(* Manages alarms *)

PROGRAM Alarm_Manager
  VAR_EXTERNAL
    Safety_OK : BOOL;
    Conveyor_Fault : BOOL;
    Mixer_Fault : BOOL;
    Packaging_Fault : BOOL;
    Pump_A_Fault : BOOL;
    Pump_B_Fault : BOOL;
    Discharge_Pump_Fault : BOOL;
    Inlet_Valve_Fault : BOOL;
    Ingredient_A_Valve_Fault : BOOL;
    Ingredient_B_Valve_Fault : BOOL;
    Discharge_Valve_Fault : BOOL;
    Batch : ST_BATCH;
    Temperature : REAL;
    Conveyor_Jam : BOOL;
    Batch_State_Code : INT;
    System_Reset : BOOL;
    Alarm_Acknowledge : BOOL;
  END_VAR
  VAR
    Safety_Alarm : ST_ALARM;
    Conveyor_Alarm : ST_ALARM;
    Mixer_Alarm : ST_ALARM;
    Packaging_Alarm : ST_ALARM;
    Pump_A_Alarm : ST_ALARM;
    Pump_B_Alarm : ST_ALARM;
    Discharge_Pump_Alarm : ST_ALARM;
    Inlet_Valve_Alarm : ST_ALARM;
    Ingredient_A_Valve_Alarm : ST_ALARM;
    Ingredient_B_Valve_Alarm : ST_ALARM;
    Discharge_Valve_Alarm : ST_ALARM;
    Conveyor_Jam_Alarm : ST_ALARM;
    Batch_Fault_Alarm : ST_ALARM;
    Temperature_Alarm : ST_ALARM;
    Any_Alarm : BOOL;
  END_VAR

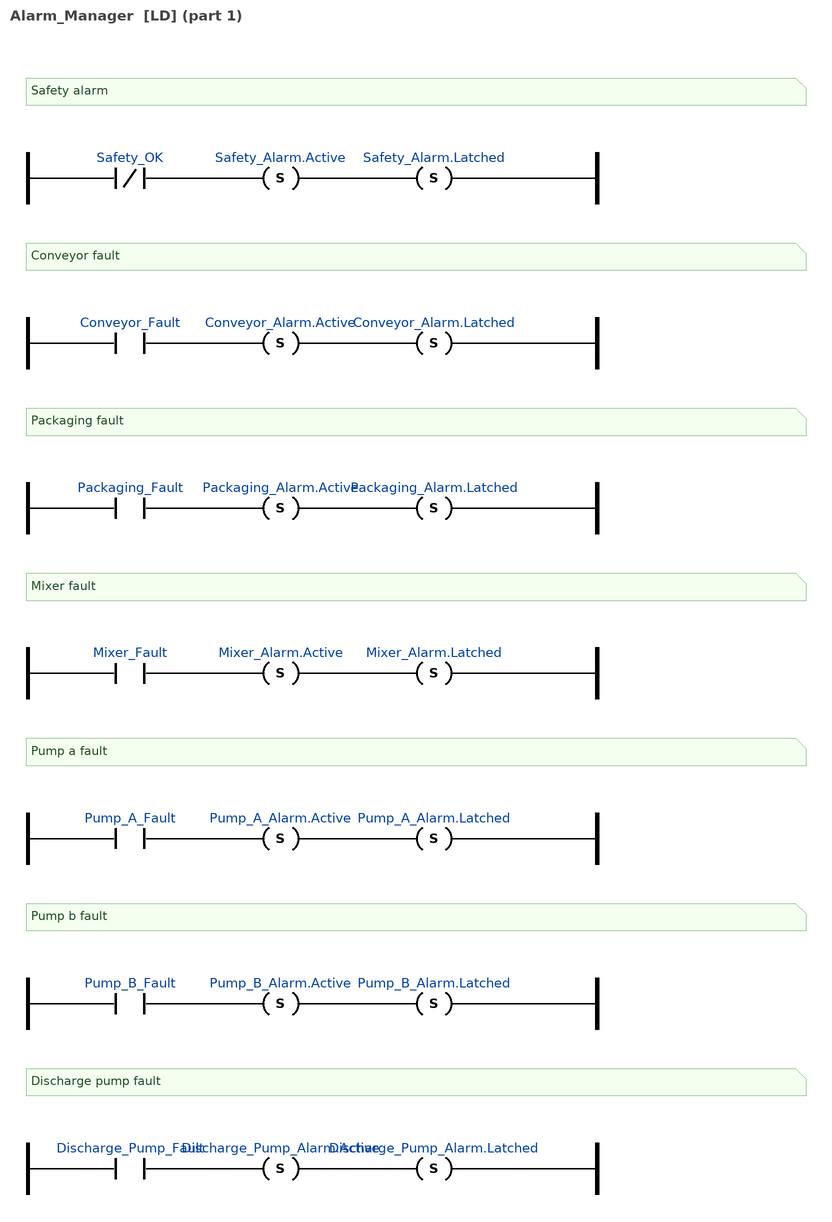
(* LD diagram, written out as Structured Text *)
(* Safety alarm *)
IF NOT Safety_OK THEN Safety_Alarm.Active := TRUE; END_IF;
IF NOT Safety_OK THEN Safety_Alarm.Latched := TRUE; END_IF;
(* Conveyor fault *)
IF Conveyor_Fault THEN Conveyor_Alarm.Active := TRUE; END_IF;
IF Conveyor_Fault THEN Conveyor_Alarm.Latched := TRUE; END_IF;
(* Packaging fault *)
IF Packaging_Fault THEN Packaging_Alarm.Active := TRUE; END_IF;
IF Packaging_Fault THEN Packaging_Alarm.Latched := TRUE; END_IF;
(* Mixer fault *)
IF Mixer_Fault THEN Mixer_Alarm.Active := TRUE; END_IF;
IF Mixer_Fault THEN Mixer_Alarm.Latched := TRUE; END_IF;
(* Pump a fault *)
IF Pump_A_Fault THEN Pump_A_Alarm.Active := TRUE; END_IF;
IF Pump_A_Fault THEN Pump_A_Alarm.Latched := TRUE; END_IF;
(* Pump b fault *)
IF Pump_B_Fault THEN Pump_B_Alarm.Active := TRUE; END_IF;
IF Pump_B_Fault THEN Pump_B_Alarm.Latched := TRUE; END_IF;
(* Discharge pump fault *)
IF Discharge_Pump_Fault THEN Discharge_Pump_Alarm.Active := TRUE; END_IF;
IF Discharge_Pump_Fault THEN Discharge_Pump_Alarm.Latched := TRUE; END_IF;
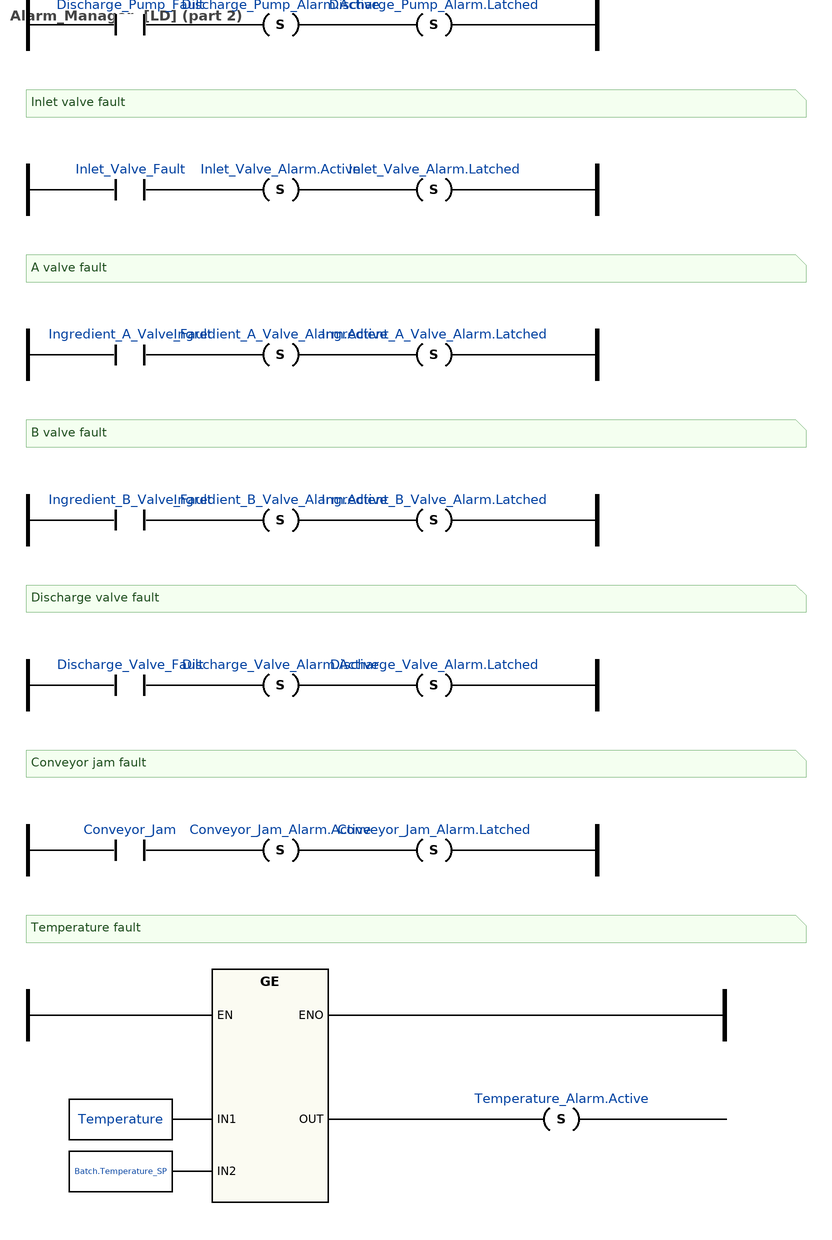
(* Inlet valve fault *)
IF Inlet_Valve_Fault THEN Inlet_Valve_Alarm.Active := TRUE; END_IF;
IF Inlet_Valve_Fault THEN Inlet_Valve_Alarm.Latched := TRUE; END_IF;
(* A valve fault *)
IF Ingredient_A_Valve_Fault THEN Ingredient_A_Valve_Alarm.Active := TRUE; END_IF;
IF Ingredient_A_Valve_Fault THEN Ingredient_A_Valve_Alarm.Latched := TRUE; END_IF;
(* B valve fault *)
IF Ingredient_B_Valve_Fault THEN Ingredient_B_Valve_Alarm.Active := TRUE; END_IF;
IF Ingredient_B_Valve_Fault THEN Ingredient_B_Valve_Alarm.Latched := TRUE; END_IF;
(* Discharge valve fault *)
IF Discharge_Valve_Fault THEN Discharge_Valve_Alarm.Active := TRUE; END_IF;
IF Discharge_Valve_Fault THEN Discharge_Valve_Alarm.Latched := TRUE; END_IF;
(* Conveyor jam fault *)
IF Conveyor_Jam THEN Conveyor_Jam_Alarm.Active := TRUE; END_IF;
IF Conveyor_Jam THEN Conveyor_Jam_Alarm.Latched := TRUE; END_IF;
(* Temperature fault *)
IF Temperature >= Batch.Temperature_SP THEN Temperature_Alarm.Active := TRUE; END_IF;
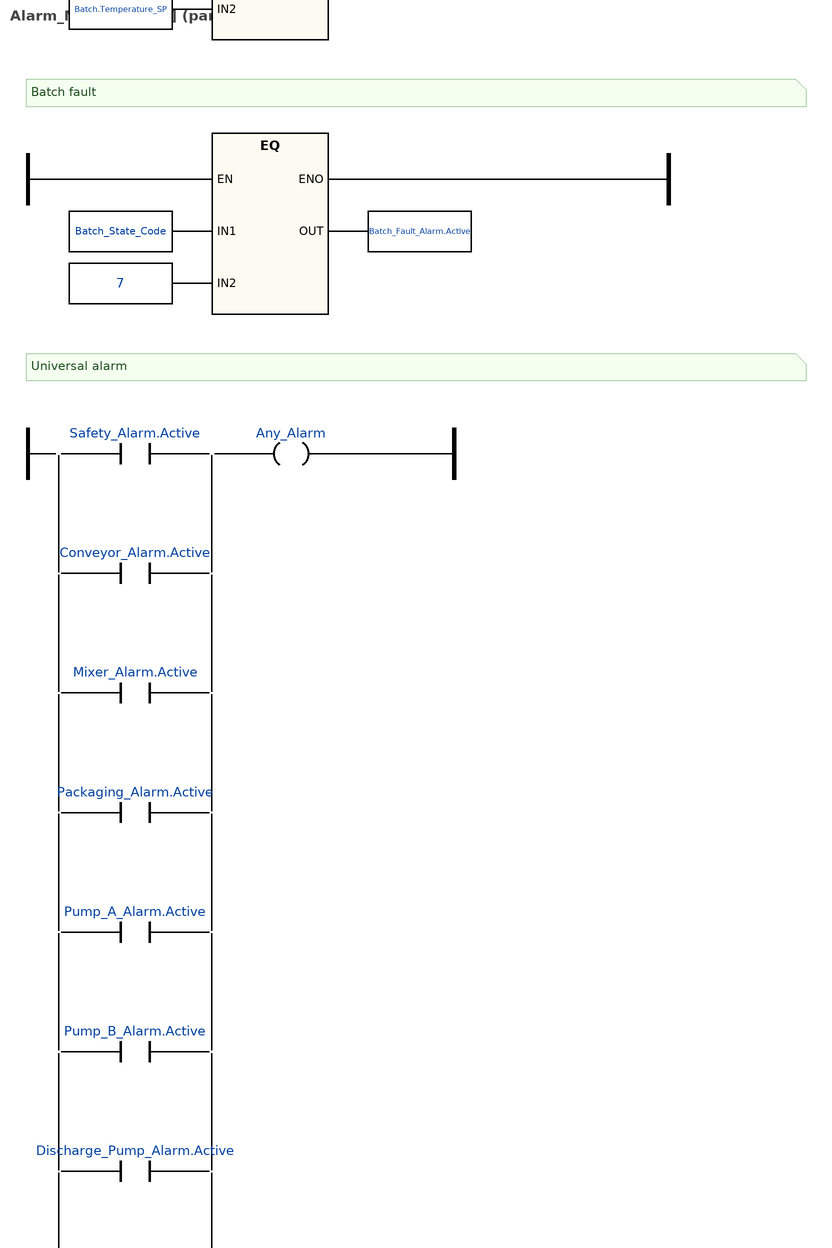
(* Batch fault *)
Batch_Fault_Alarm.Active := Batch_State_Code = 7;
(* Universal alarm *)
Any_Alarm := Safety_Alarm.Active OR Conveyor_Alarm.Active OR Mixer_Alarm.Active OR Packaging_Alarm.Active OR Pump_A_Alarm.Active OR Pump_B_Alarm.Active OR Discharge_Pump_Alarm.Active OR Inlet_Valve_Alarm.Active OR Ingredient_A_Valve_Alarm.Active OR Ingredient_B_Valve_Alarm.Active OR Discharge_Valve_Alarm.Active OR Conveyor_Jam_Alarm.Active OR Batch_Fault_Alarm.Active OR Temperature_Alarm.Active;
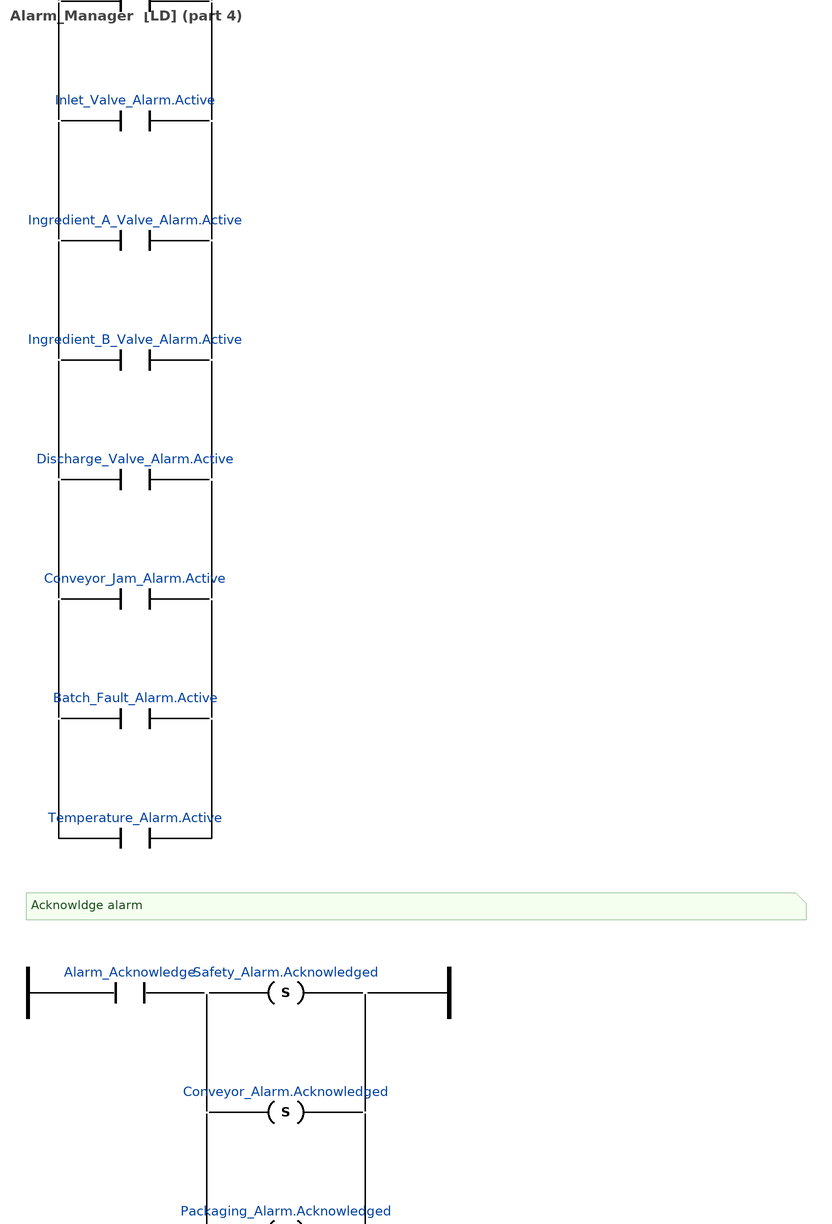
(* Acknowldge alarm *)
IF Alarm_Acknowledge THEN Safety_Alarm.Acknowledged := TRUE; END_IF;
IF Alarm_Acknowledge THEN Conveyor_Alarm.Acknowledged := TRUE; END_IF;
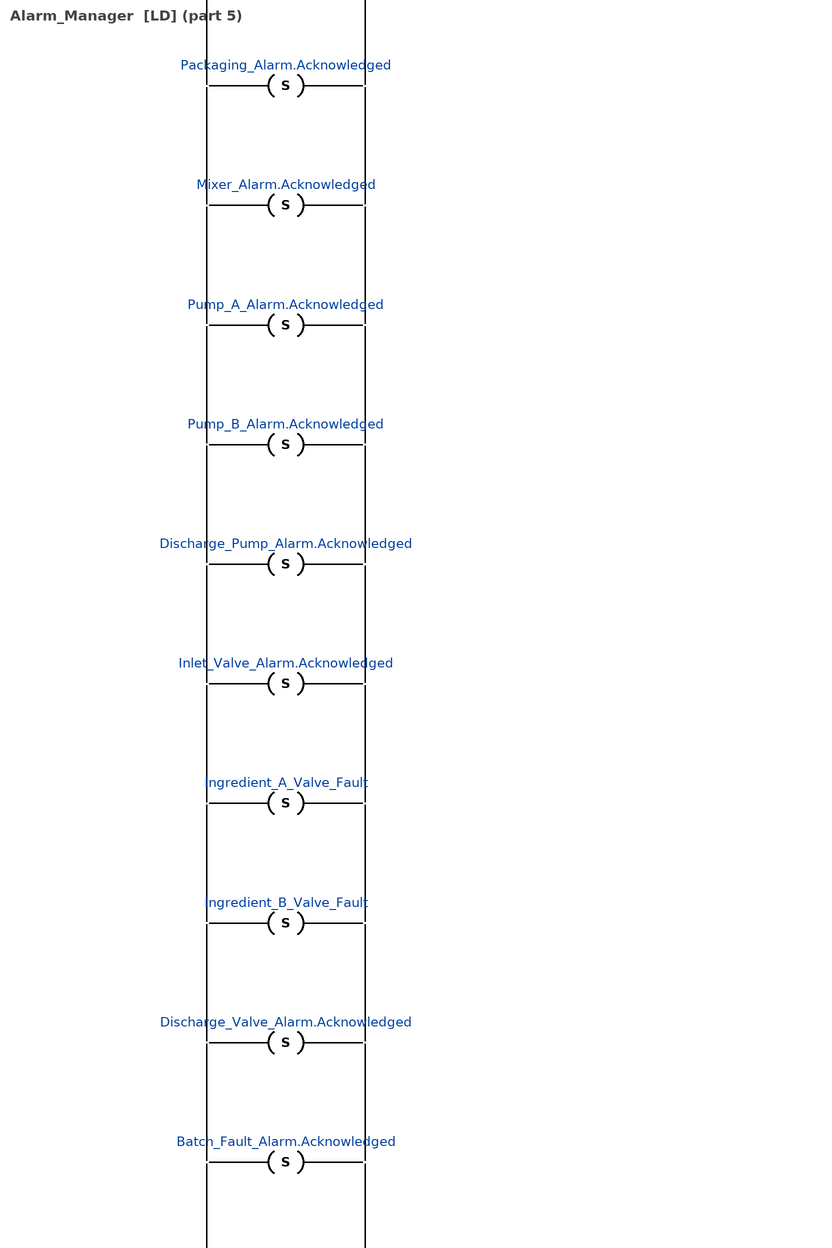
IF Alarm_Acknowledge THEN Packaging_Alarm.Acknowledged := TRUE; END_IF;
IF Alarm_Acknowledge THEN Mixer_Alarm.Acknowledged := TRUE; END_IF;
IF Alarm_Acknowledge THEN Pump_A_Alarm.Acknowledged := TRUE; END_IF;
IF Alarm_Acknowledge THEN Pump_B_Alarm.Acknowledged := TRUE; END_IF;
IF Alarm_Acknowledge THEN Discharge_Pump_Alarm.Acknowledged := TRUE; END_IF;
IF Alarm_Acknowledge THEN Inlet_Valve_Alarm.Acknowledged := TRUE; END_IF;
IF Alarm_Acknowledge THEN Ingredient_A_Valve_Fault := TRUE; END_IF;
IF Alarm_Acknowledge THEN Ingredient_B_Valve_Fault := TRUE; END_IF;
IF Alarm_Acknowledge THEN Discharge_Valve_Alarm.Acknowledged := TRUE; END_IF;
IF Alarm_Acknowledge THEN Batch_Fault_Alarm.Acknowledged := TRUE; END_IF;
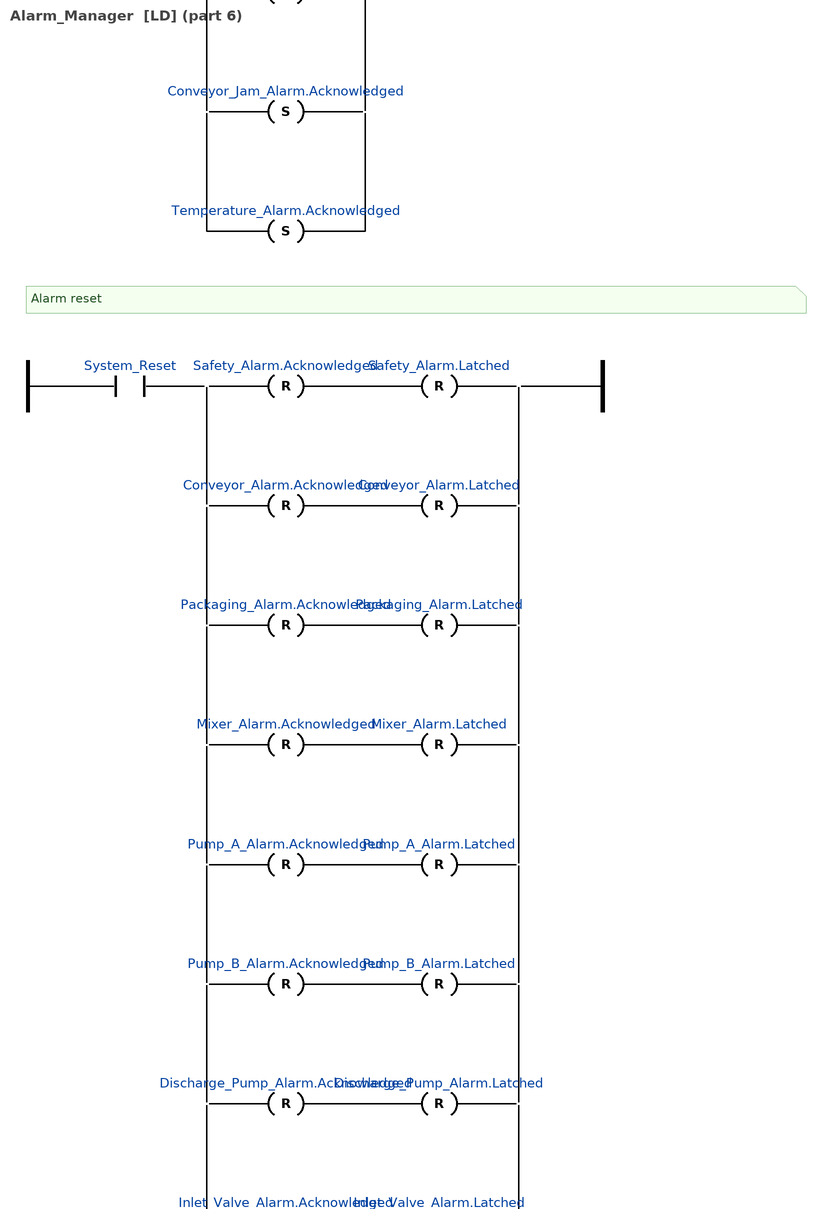
IF Alarm_Acknowledge THEN Conveyor_Jam_Alarm.Acknowledged := TRUE; END_IF;
IF Alarm_Acknowledge THEN Temperature_Alarm.Acknowledged := TRUE; END_IF;
(* Alarm reset *)
IF System_Reset THEN Safety_Alarm.Acknowledged := FALSE; END_IF;
IF System_Reset THEN Safety_Alarm.Latched := FALSE; END_IF;
IF System_Reset THEN Conveyor_Alarm.Acknowledged := FALSE; END_IF;
IF System_Reset THEN Conveyor_Alarm.Latched := FALSE; END_IF;
IF System_Reset THEN Packaging_Alarm.Acknowledged := FALSE; END_IF;
IF System_Reset THEN Packaging_Alarm.Latched := FALSE; END_IF;
IF System_Reset THEN Mixer_Alarm.Acknowledged := FALSE; END_IF;
IF System_Reset THEN Mixer_Alarm.Latched := FALSE; END_IF;
IF System_Reset THEN Pump_A_Alarm.Acknowledged := FALSE; END_IF;
IF System_Reset THEN Pump_A_Alarm.Latched := FALSE; END_IF;
IF System_Reset THEN Pump_B_Alarm.Acknowledged := FALSE; END_IF;
IF System_Reset THEN Pump_B_Alarm.Latched := FALSE; END_IF;
IF System_Reset THEN Discharge_Pump_Alarm.Acknowledged := FALSE; END_IF;
IF System_Reset THEN Discharge_Pump_Alarm.Latched := FALSE; END_IF;
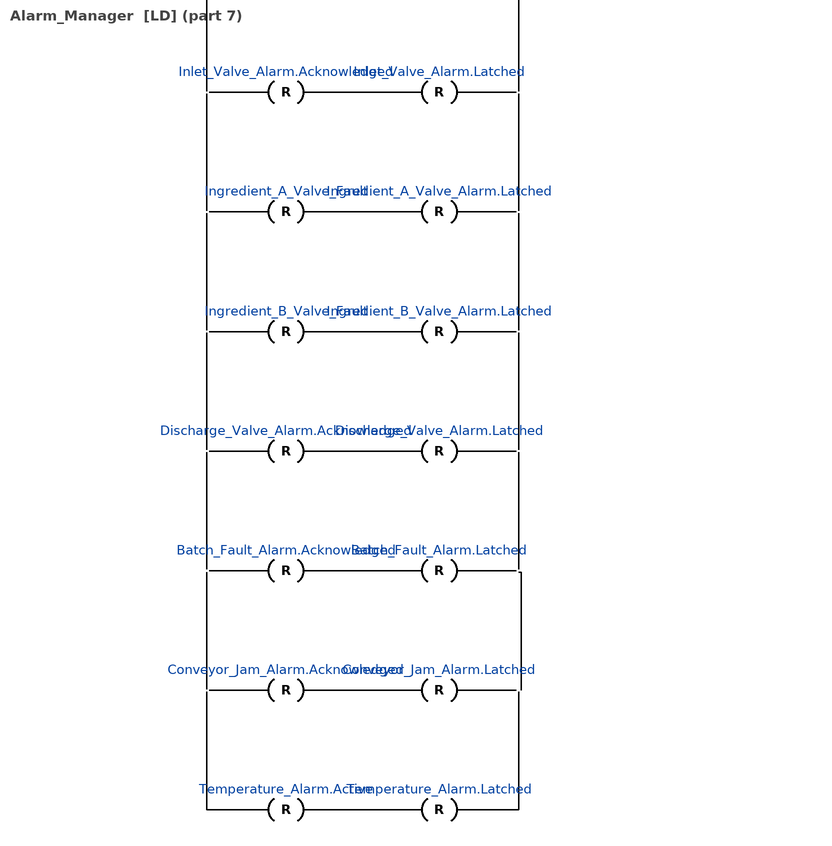
IF System_Reset THEN Inlet_Valve_Alarm.Acknowledged := FALSE; END_IF;
IF System_Reset THEN Inlet_Valve_Alarm.Latched := FALSE; END_IF;
IF System_Reset THEN Ingredient_A_Valve_Fault := FALSE; END_IF;
IF System_Reset THEN Ingredient_A_Valve_Alarm.Latched := FALSE; END_IF;
IF System_Reset THEN Ingredient_B_Valve_Fault := FALSE; END_IF;
IF System_Reset THEN Ingredient_B_Valve_Alarm.Latched := FALSE; END_IF;
IF System_Reset THEN Discharge_Valve_Alarm.Acknowledged := FALSE; END_IF;
IF System_Reset THEN Discharge_Valve_Alarm.Latched := FALSE; END_IF;
IF System_Reset THEN Batch_Fault_Alarm.Acknowledged := FALSE; END_IF;
IF System_Reset THEN Batch_Fault_Alarm.Latched := FALSE; END_IF;
IF System_Reset THEN Conveyor_Jam_Alarm.Acknowledged := FALSE; END_IF;
IF System_Reset THEN Conveyor_Jam_Alarm.Latched := FALSE; END_IF;
IF System_Reset THEN Temperature_Alarm.Active := FALSE; END_IF;
IF System_Reset THEN Temperature_Alarm.Latched := FALSE; END_IF;
END_PROGRAM
